FUNCTION AddRPS : RobotPoseSimple
VAR_INPUT
	pose1, pose2: RobotPoseSimple;
END_VAR
VAR
END_VAR

AddRPS.x		:= pose1.x + pose2.x;
AddRPS.y		:= pose1.y + pose2.y;
AddRPS.theta	:= pose1.theta + pose2.theta;

END_FUNCTION

(* stored: Version 1.1.0.1, ProductVersion 3.1.4024.11
   POU AddRPS: Id {68a1e610-742f-4602-90ea-14eef65fa4c1}, SpecialFunc None *)
